TYPE ST_ORCA_SiteInfo :
STRUCT

	ProductionSite 			: STRING(255);
	ProductionLine 		: STRING(255);


END_STRUCT
END_TYPE

(* stored: Version 1.1.0.1
   DUT ST_ORCA_SiteInfo: Id {1a92788f-f2dd-42b7-955c-42ed84d7e29a} *)
